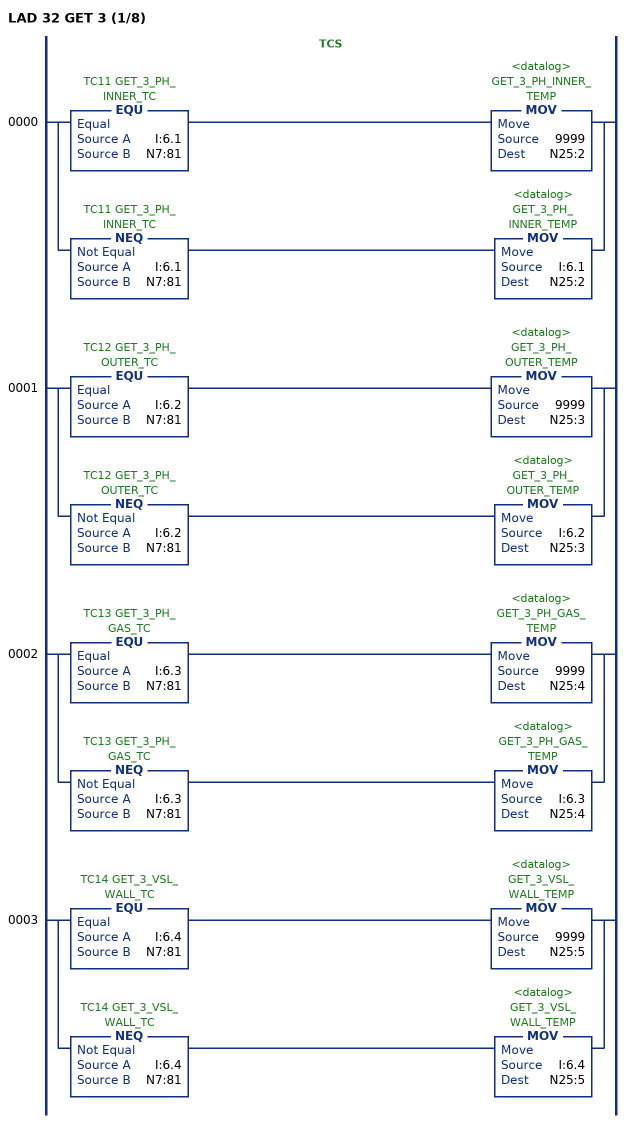
% Rung: 0 %
% TITLE: TCS %
SOR BST EQU I:6.1 N7:81 MOV 9999 N25:2 NXB NEQ I:6.1 N7:81 MOV I:6.1 N25:2 BND EOR
%   I:6.1  GET_3_PH_INNER_TC  "TC11" %
%   N7:81  TC_OPEN_SP  "CONFIG The value read by an open TC input" %
%   N25:2  GET_3_PH_INNER_TEMP  "<datalog>" %
% Rung: 1 %
SOR BST EQU I:6.2 N7:81 MOV 9999 N25:3 NXB NEQ I:6.2 N7:81 MOV I:6.2 N25:3 BND EOR
%   I:6.2  GET_3_PH_OUTER_TC  "TC12" %
%   N7:81  TC_OPEN_SP  "CONFIG The value read by an open TC input" %
%   N25:3  GET_3_PH_OUTER_TEMP  "<datalog>" %
% Rung: 2 %
SOR BST EQU I:6.3 N7:81 MOV 9999 N25:4 NXB NEQ I:6.3 N7:81 MOV I:6.3 N25:4 BND EOR
%   I:6.3  GET_3_PH_GAS_TC  "TC13" %
%   N7:81  TC_OPEN_SP  "CONFIG The value read by an open TC input" %
%   N25:4  GET_3_PH_GAS_TEMP  "<datalog>" %
% Rung: 3 %
SOR BST EQU I:6.4 N7:81 MOV 9999 N25:5 NXB NEQ I:6.4 N7:81 MOV I:6.4 N25:5 BND EOR
%   I:6.4  GET_3_VSL_WALL_TC  "TC14" %
%   N7:81  TC_OPEN_SP  "CONFIG The value read by an open TC input" %
%   N25:5  GET_3_VSL_WALL_TEMP  "<datalog>" %

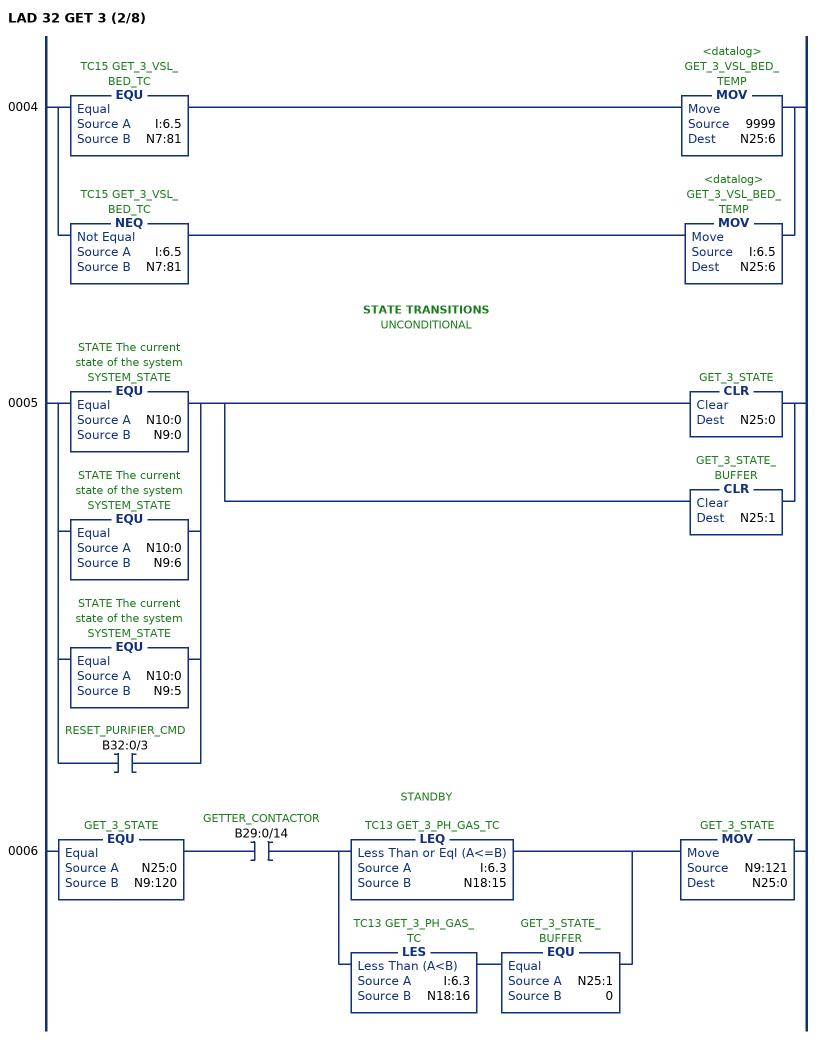
% Rung: 4 %
SOR BST EQU I:6.5 N7:81 MOV 9999 N25:6 NXB NEQ I:6.5 N7:81 MOV I:6.5 N25:6 BND EOR
%   I:6.5  GET_3_VSL_BED_TC  "TC15" %
%   N7:81  TC_OPEN_SP  "CONFIG The value read by an open TC input" %
%   N25:6  GET_3_VSL_BED_TEMP  "<datalog>" %
% Rung: 5 %
% TITLE: STATE TRANSITIONS %
% UNCONDITIONAL %
SOR BST EQU N10:0 N9:0 NXB EQU N10:0 N9:6 NXB EQU N10:0 N9:5 NXB XIC B32:0/3 BND BST CLR N25:0 NXB CLR N25:1 BND EOR
%   N10:0  SYSTEM_STATE  "STATE The current state of the system" %
%   N9:0  SYSTEM_OFFLINE %
%   N9:6  SYSTEM_PURGE %
%   N9:5  SYSTEM_QUICK_START %
%   B32:0/3  RESET_PURIFIER_CMD %
%   N25:0  GET_3_STATE %
%   N25:1  GET_3_STATE_BUFFER %
% Rung: 6 %
% STANDBY %
SOR EQU N25:0 N9:120 XIC B29:0/14 BST LEQ I:6.3 N18:15 NXB LES I:6.3 N18:16 EQU N25:1 0 BND MOV N9:121 N25:0 EOR
%   N25:0  GET_3_STATE %
%   N9:120  GETTER_STANDBY %
%   B29:0/14  GETTER_CONTACTOR %
%   I:6.3  GET_3_PH_GAS_TC  "TC13" %
%   N18:15  GETTER_SS_BEGIN_TEMP %
%   N18:16  GETTER_SS_END_TEMP %
%   N25:1  GET_3_STATE_BUFFER %
%   N9:121  GETTER_SOFTSTART %

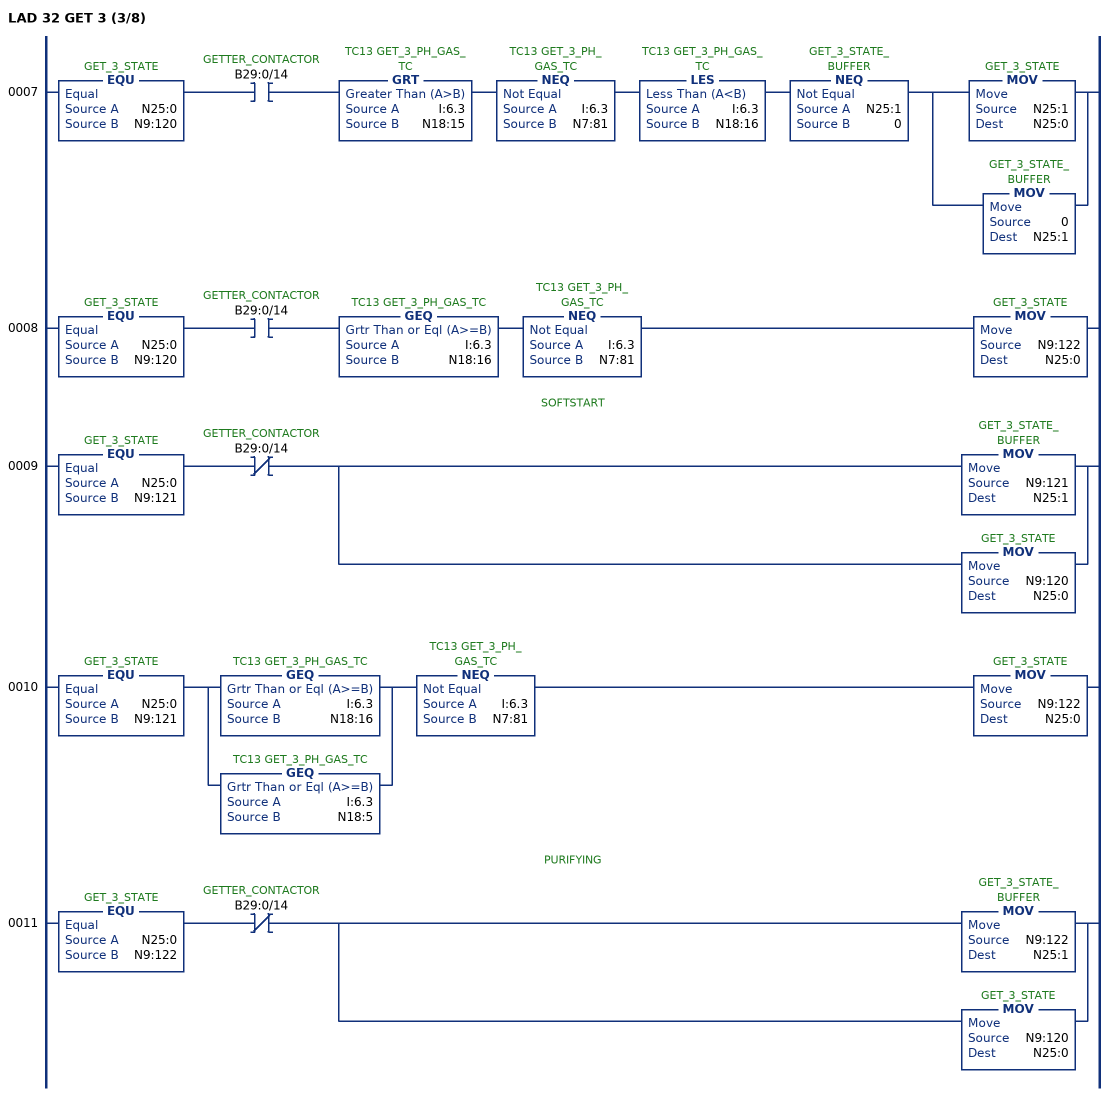
% Rung: 7 %
SOR EQU N25:0 N9:120 XIC B29:0/14 GRT I:6.3 N18:15 NEQ I:6.3 N7:81 LES I:6.3 N18:16 NEQ N25:1 0 BST MOV N25:1 N25:0 NXB MOV 0 N25:1 BND EOR
%   N25:0  GET_3_STATE %
%   N9:120  GETTER_STANDBY %
%   B29:0/14  GETTER_CONTACTOR %
%   I:6.3  GET_3_PH_GAS_TC  "TC13" %
%   N18:15  GETTER_SS_BEGIN_TEMP %
%   N7:81  TC_OPEN_SP  "CONFIG The value read by an open TC input" %
%   N18:16  GETTER_SS_END_TEMP %
%   N25:1  GET_3_STATE_BUFFER %
% Rung: 8 %
SOR EQU N25:0 N9:120 XIC B29:0/14 GEQ I:6.3 N18:16 NEQ I:6.3 N7:81 MOV N9:122 N25:0 EOR
%   N25:0  GET_3_STATE %
%   N9:120  GETTER_STANDBY %
%   B29:0/14  GETTER_CONTACTOR %
%   I:6.3  GET_3_PH_GAS_TC  "TC13" %
%   N18:16  GETTER_SS_END_TEMP %
%   N7:81  TC_OPEN_SP  "CONFIG The value read by an open TC input" %
%   N9:122  GETTER_PURIFYING %
% Rung: 9 %
% SOFTSTART %
SOR EQU N25:0 N9:121 XIO B29:0/14 BST MOV N9:121 N25:1 NXB MOV N9:120 N25:0 BND EOR
%   N25:0  GET_3_STATE %
%   N9:121  GETTER_SOFTSTART %
%   B29:0/14  GETTER_CONTACTOR %
%   N25:1  GET_3_STATE_BUFFER %
%   N9:120  GETTER_STANDBY %
% Rung: 10 %
SOR EQU N25:0 N9:121 BST GEQ I:6.3 N18:16 NXB GEQ I:6.3 N18:5 BND NEQ I:6.3 N7:81 MOV N9:122 N25:0 EOR
%   N25:0  GET_3_STATE %
%   N9:121  GETTER_SOFTSTART %
%   I:6.3  GET_3_PH_GAS_TC  "TC13" %
%   N18:16  GETTER_SS_END_TEMP %
%   N18:5  GETTER_PH_SP  "<datalog>" %
%   N7:81  TC_OPEN_SP  "CONFIG The value read by an open TC input" %
%   N9:122  GETTER_PURIFYING %
% Rung: 11 %
% PURIFYING %
SOR EQU N25:0 N9:122 XIO B29:0/14 BST MOV N9:122 N25:1 NXB MOV N9:120 N25:0 BND EOR
%   N25:0  GET_3_STATE %
%   N9:122  GETTER_PURIFYING %
%   B29:0/14  GETTER_CONTACTOR %
%   N25:1  GET_3_STATE_BUFFER %
%   N9:120  GETTER_STANDBY %

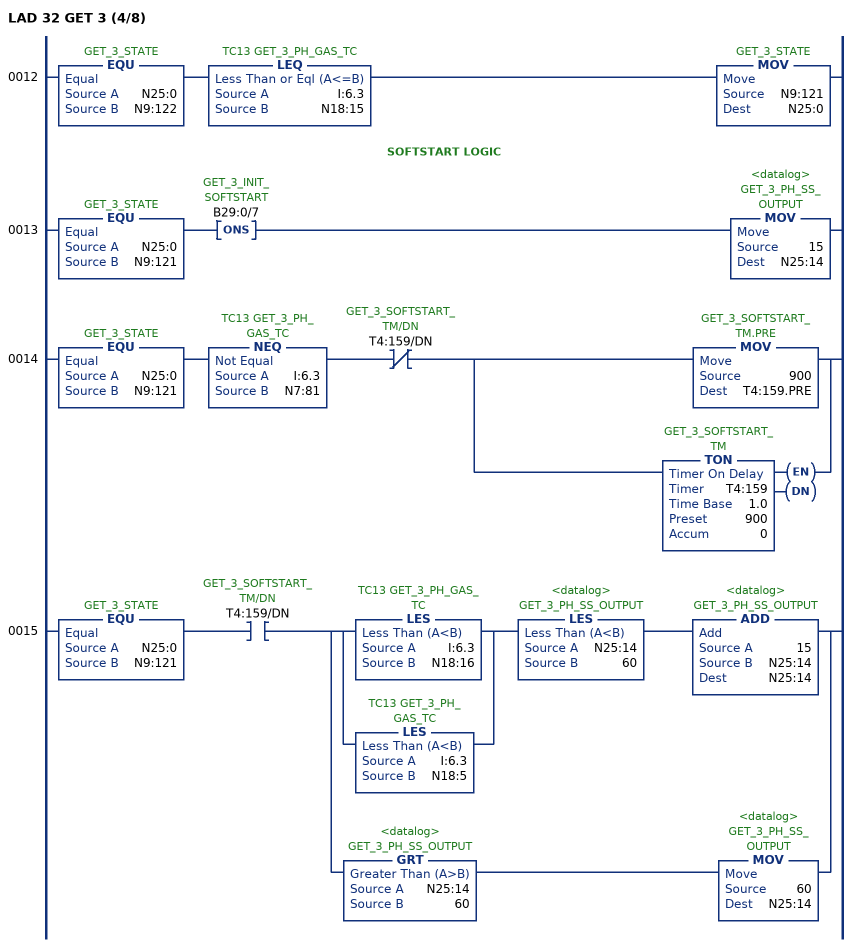
% Rung: 12 %
SOR EQU N25:0 N9:122 LEQ I:6.3 N18:15 MOV N9:121 N25:0 EOR
%   N25:0  GET_3_STATE %
%   N9:122  GETTER_PURIFYING %
%   I:6.3  GET_3_PH_GAS_TC  "TC13" %
%   N18:15  GETTER_SS_BEGIN_TEMP %
%   N9:121  GETTER_SOFTSTART %
% Rung: 13 %
% TITLE: SOFTSTART LOGIC %
SOR EQU N25:0 N9:121 ONS B29:0/7 MOV 15 N25:14 EOR
%   N25:0  GET_3_STATE %
%   N9:121  GETTER_SOFTSTART %
%   B29:0/7  GET_3_INIT_SOFTSTART %
%   N25:14  GET_3_PH_SS_OUTPUT  "<datalog>" %
% Rung: 14 %
SOR EQU N25:0 N9:121 NEQ I:6.3 N7:81 XIO T4:159/DN BST MOV 900 T4:159.PRE NXB TON T4:159 1.0 900 0 BND EOR
%   N25:0  GET_3_STATE %
%   N9:121  GETTER_SOFTSTART %
%   I:6.3  GET_3_PH_GAS_TC  "TC13" %
%   N7:81  TC_OPEN_SP  "CONFIG The value read by an open TC input" %
%   T4:159  GET_3_SOFTSTART_TM %
% Rung: 15 %
SOR EQU N25:0 N9:121 XIC T4:159/DN BST BST LES I:6.3 N18:16 NXB LES I:6.3 N18:5 BND LES N25:14 60 ADD 15 N25:14 N25:14 NXB GRT N25:14 60 MOV 60 N25:14 BND EOR
%   N25:0  GET_3_STATE %
%   N9:121  GETTER_SOFTSTART %
%   T4:159  GET_3_SOFTSTART_TM %
%   I:6.3  GET_3_PH_GAS_TC  "TC13" %
%   N18:16  GETTER_SS_END_TEMP %
%   N18:5  GETTER_PH_SP  "<datalog>" %
%   N25:14  GET_3_PH_SS_OUTPUT  "<datalog>" %

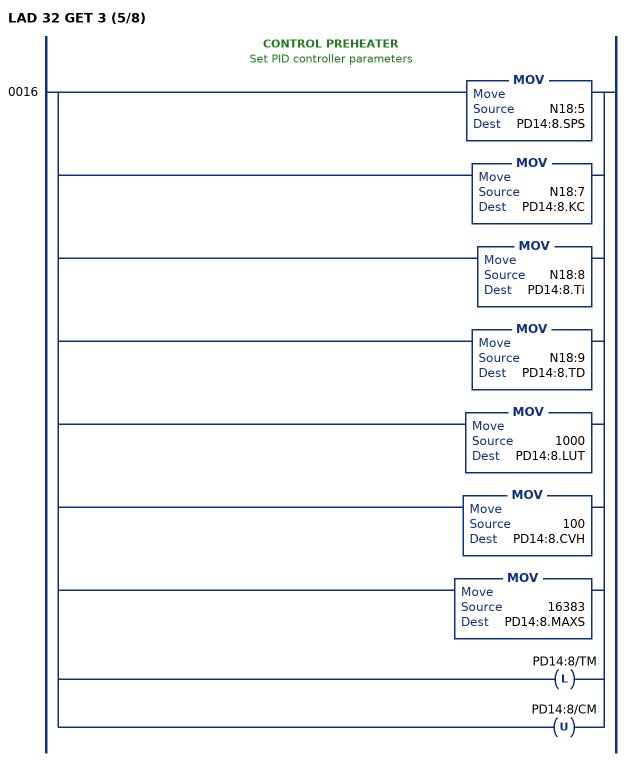
% Rung: 16 %
% TITLE: CONTROL PREHEATER %
% Set PID controller parameters %
SOR BST MOV N18:5 PD14:8.SPS NXB MOV N18:7 PD14:8.KC NXB MOV N18:8 PD14:8.Ti NXB MOV N18:9 PD14:8.TD NXB MOV 1000 PD14:8.LUT NXB MOV 100 PD14:8.CVH NXB MOV 16383 PD14:8.MAXS NXB OTL PD14:8/TM NXB OTU PD14:8/CM BND EOR
%   N18:5  GETTER_PH_SP  "<datalog>" %
%   N18:7  GET_PH_PID_GAIN %
%   N18:8  GET_PH_PID_INTEG %
%   N18:9  GET_PH_PID_DERIV %

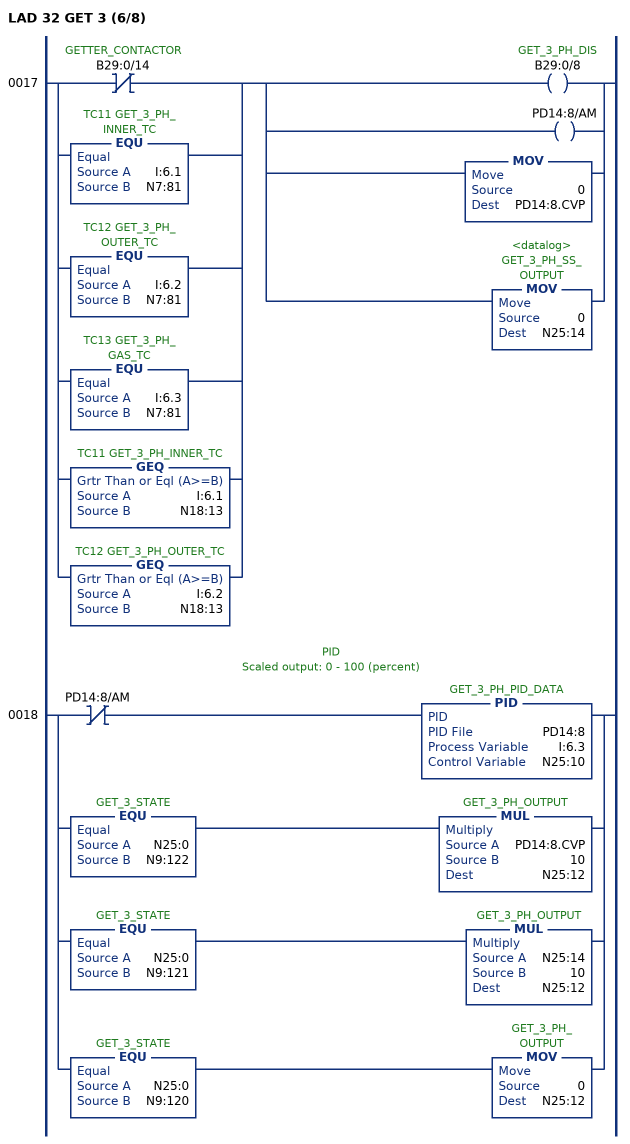
% Rung: 17 %
SOR BST XIO B29:0/14 NXB EQU I:6.1 N7:81 NXB EQU I:6.2 N7:81 NXB EQU I:6.3 N7:81 NXB GEQ I:6.1 N18:13 NXB GEQ I:6.2 N18:13 BND BST OTE B29:0/8 NXB OTE PD14:8/AM NXB MOV 0 PD14:8.CVP NXB MOV 0 N25:14 BND EOR
%   B29:0/14  GETTER_CONTACTOR %
%   I:6.1  GET_3_PH_INNER_TC  "TC11" %
%   N7:81  TC_OPEN_SP  "CONFIG The value read by an open TC input" %
%   I:6.2  GET_3_PH_OUTER_TC  "TC12" %
%   I:6.3  GET_3_PH_GAS_TC  "TC13" %
%   N18:13  GET_PH_ROD_LIMIT %
%   B29:0/8  GET_3_PH_DIS %
%   N25:14  GET_3_PH_SS_OUTPUT  "<datalog>" %
% Rung: 18 %
% PID
% Scaled output: 0 - 100 (percent) %
SOR BST XIO PD14:8/AM PID PD14:8 I:6.3 N25:10 NXB EQU N25:0 N9:122 MUL PD14:8.CVP 10 N25:12 NXB EQU N25:0 N9:121 MUL N25:14 10 N25:12 NXB EQU N25:0 N9:120 MOV 0 N25:12 BND EOR
%   PD14:8  GET_3_PH_PID_DATA %
%   I:6.3  GET_3_PH_GAS_TC  "TC13" %
%   N25:10  GET_3_PH_OUT_RAW %
%   N25:0  GET_3_STATE %
%   N9:122  GETTER_PURIFYING %
%   N25:12  GET_3_PH_OUTPUT %
%   N9:121  GETTER_SOFTSTART %
%   N25:14  GET_3_PH_SS_OUTPUT  "<datalog>" %
%   N9:120  GETTER_STANDBY %

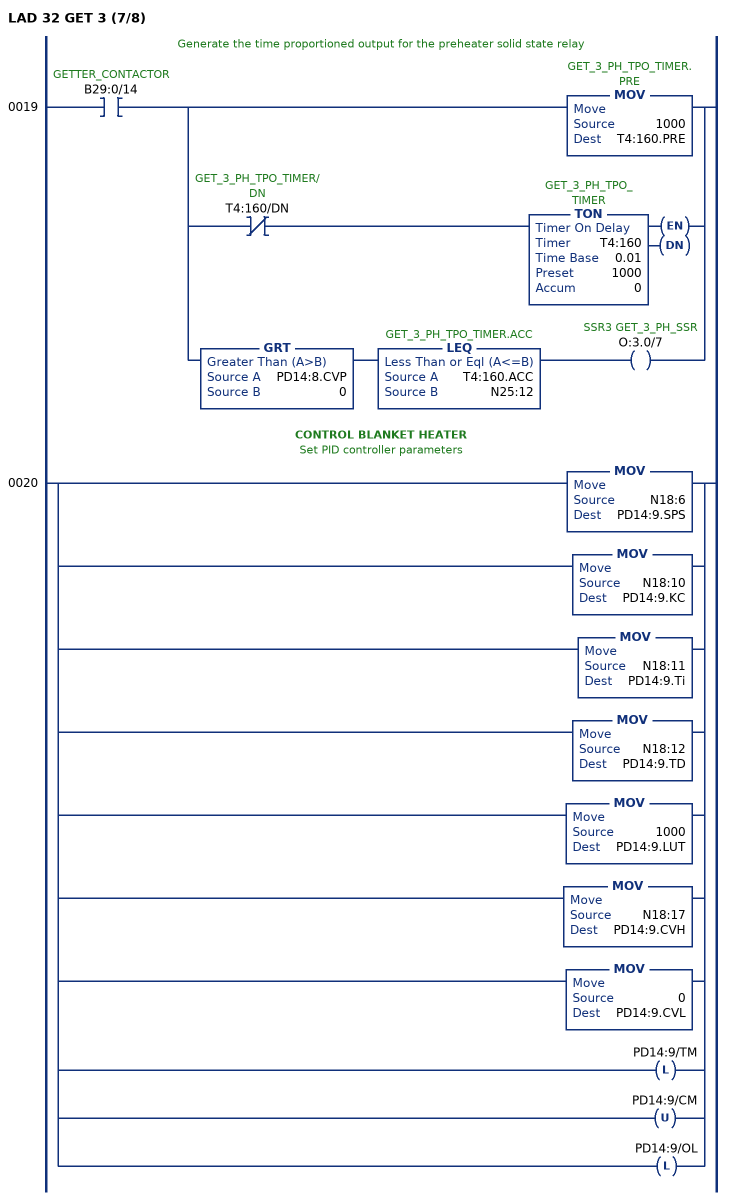
% Rung: 19 %
% Generate the time proportioned output for the preheater solid state relay %
SOR XIC B29:0/14 BST MOV 1000 T4:160.PRE NXB XIO T4:160/DN TON T4:160 0.01 1000 0 NXB GRT PD14:8.CVP 0 LEQ T4:160.ACC N25:12 OTE O:3.0/7 BND EOR
%   B29:0/14  GETTER_CONTACTOR %
%   T4:160  GET_3_PH_TPO_TIMER %
%   N25:12  GET_3_PH_OUTPUT %
%   O:3.0/7  GET_3_PH_SSR  "SSR3" %
% Rung: 20 %
% TITLE: CONTROL BLANKET HEATER %
% Set PID controller parameters %
SOR BST MOV N18:6 PD14:9.SPS NXB MOV N18:10 PD14:9.KC NXB MOV N18:11 PD14:9.Ti NXB MOV N18:12 PD14:9.TD NXB MOV 1000 PD14:9.LUT NXB MOV N18:17 PD14:9.CVH NXB MOV 0 PD14:9.CVL NXB OTL PD14:9/TM NXB OTU PD14:9/CM NXB OTL PD14:9/OL BND EOR
%   N18:6  GETTER_BLKT_SP  "<datalog>" %
%   N18:10  GET_BLKT_PID_GAIN %
%   N18:11  GET_BLKT_PID_INTEG %
%   N18:12  GET_BLKT_PID_DERIV %
%   N18:17  GET_BLKT_PID_HI_LIM %

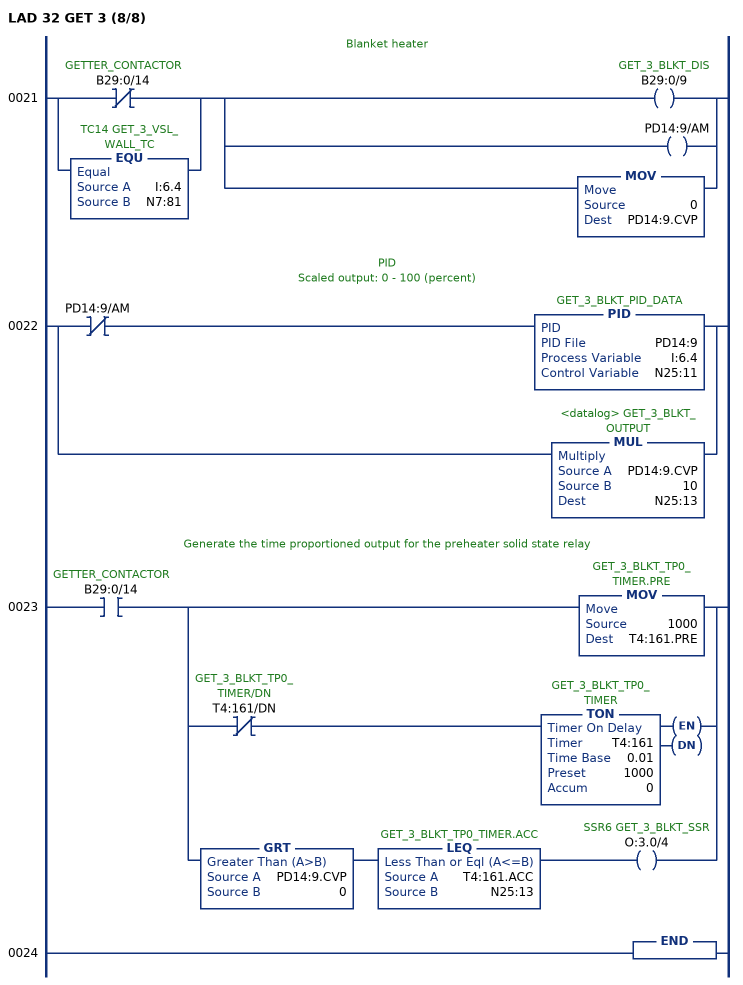
% Rung: 21 %
% Blanket heater %
SOR BST XIO B29:0/14 NXB EQU I:6.4 N7:81 BND BST OTE B29:0/9 NXB OTE PD14:9/AM NXB MOV 0 PD14:9.CVP BND EOR
%   B29:0/14  GETTER_CONTACTOR %
%   I:6.4  GET_3_VSL_WALL_TC  "TC14" %
%   N7:81  TC_OPEN_SP  "CONFIG The value read by an open TC input" %
%   B29:0/9  GET_3_BLKT_DIS %
% Rung: 22 %
% PID
% Scaled output: 0 - 100 (percent) %
SOR BST XIO PD14:9/AM PID PD14:9 I:6.4 N25:11 NXB MUL PD14:9.CVP 10 N25:13 BND EOR
%   PD14:9  GET_3_BLKT_PID_DATA %
%   I:6.4  GET_3_VSL_WALL_TC  "TC14" %
%   N25:11  GET_3_BLKT_OUT_RAW %
%   N25:13  GET_3_BLKT_OUTPUT  "<datalog>" %
% Rung: 23 %
% Generate the time proportioned output for the preheater solid state relay %
SOR XIC B29:0/14 BST MOV 1000 T4:161.PRE NXB XIO T4:161/DN TON T4:161 0.01 1000 0 NXB GRT PD14:9.CVP 0 LEQ T4:161.ACC N25:13 OTE O:3.0/4 BND EOR
%   B29:0/14  GETTER_CONTACTOR %
%   T4:161  GET_3_BLKT_TP0_TIMER %
%   N25:13  GET_3_BLKT_OUTPUT  "<datalog>" %
%   O:3.0/4  GET_3_BLKT_SSR  "SSR6" %
% Rung: 24 %
SOR END EOR

LADDER 49 "MODBUS"
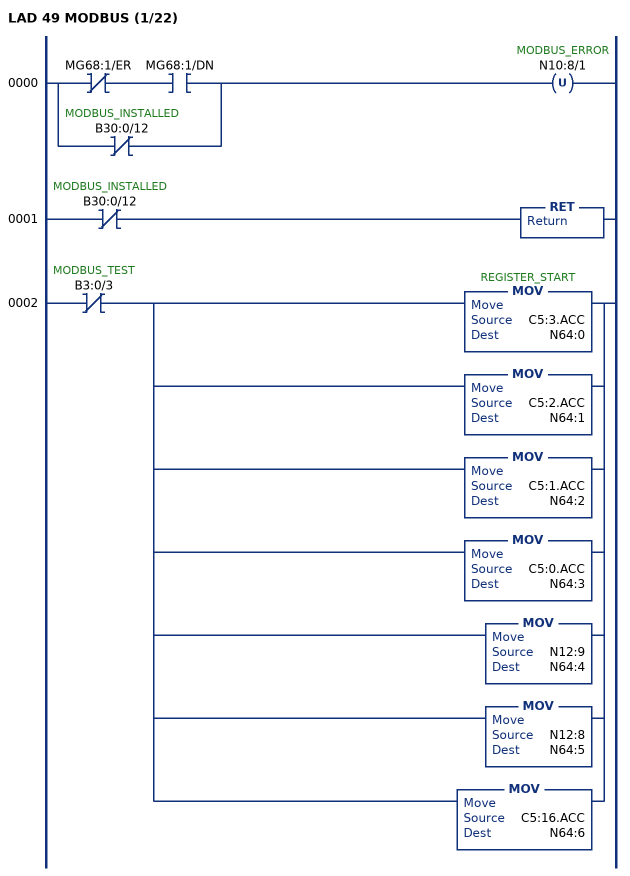
% Rung: 0 %
SOR BST XIO MG68:1/ER XIC MG68:1/DN NXB XIO B30:0/12 BND OTU N10:8/1 EOR
%   B30:0/12  MODBUS_INSTALLED %
%   N10:8/1  MODBUS_ERROR %
% Rung: 1 %
SOR XIO B30:0/12 RET EOR
%   B30:0/12  MODBUS_INSTALLED %
% Rung: 2 %
SOR XIO B3:0/3 BST MOV C5:3.ACC N64:0 NXB MOV C5:2.ACC N64:1 NXB MOV C5:1.ACC N64:2 NXB MOV C5:0.ACC N64:3 NXB MOV N12:9 N64:4 NXB MOV N12:8 N64:5 NXB MOV C5:16.ACC N64:6 BND EOR
%   B3:0/3  MODBUS_TEST %
%   C5:3  PURIFY_ACTIVE_TTL_DY  "COUNTER The number of total elapsed purification days for the process equipment" %
%   N64:0  REGISTER_START %
%   C5:2  PURIFY_ACTIVE_TTL_HR  "COUNTER The number of total elapsed purification hours for the process equipment" %
%   C5:1  PURIFY_ACTIVE_MINUTE  "COUNTER The number of elapsed purification minutes for the current ADS (60 min)" %
%   C5:0  PURIFY_ACTIVE_HOURS  "COUNTER The number of elapsed purification hours for the current ADS" %
%   N12:9  MIN_LEFT_IN_PURIFY %
%   N12:8  HRS_LEFT_IN_PURIFY %
%   C5:16  GETTER_SERVICE_DAYS %

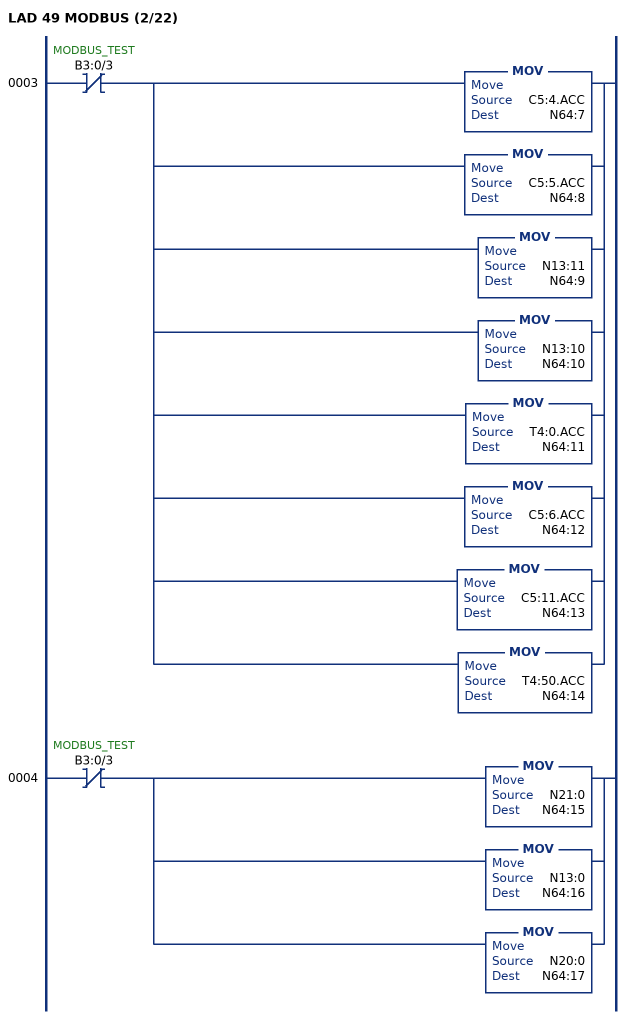
% Rung: 3 %
SOR XIO B3:0/3 BST MOV C5:4.ACC N64:7 NXB MOV C5:5.ACC N64:8 NXB MOV N13:11 N64:9 NXB MOV N13:10 N64:10 NXB MOV T4:0.ACC N64:11 NXB MOV C5:6.ACC N64:12 NXB MOV C5:11.ACC N64:13 NXB MOV T4:50.ACC N64:14 BND EOR
%   B3:0/3  MODBUS_TEST %
%   C5:4  REGEN_RUN_MINUTE %
%   C5:5  REGEN_COOL_MINUTE  "COUNTER Regen the number of minutes for which the bed has cooled" %
%   N13:11  REGEN_MIN_LEFT  "STATUS Preheater Alarm Measured temperature change" %
%   N13:10  REGEN_HRS_LEFT  "STATUS Regen Preheater Temperature Initial Temperature" %
%   T4:0  PURIFY_OVERLAP_TIMER  "TIMER Purify Overlap" %
%   C5:6  START_PURGE_CTR %
%   C5:11  H2_LEAK_RST_MIN %
%   T4:50  H2_LEAK_RST_SEC %
% Rung: 4 %
SOR XIO B3:0/3 BST MOV N21:0 N64:15 NXB MOV N13:0 N64:16 NXB MOV N20:0 N64:17 BND EOR
%   B3:0/3  MODBUS_TEST %
%   N21:0  START_STATE %
%   N13:0  REGEN_STATE  "STATE The current state of the regen process" %
%   N20:0  PURGE_STATE %

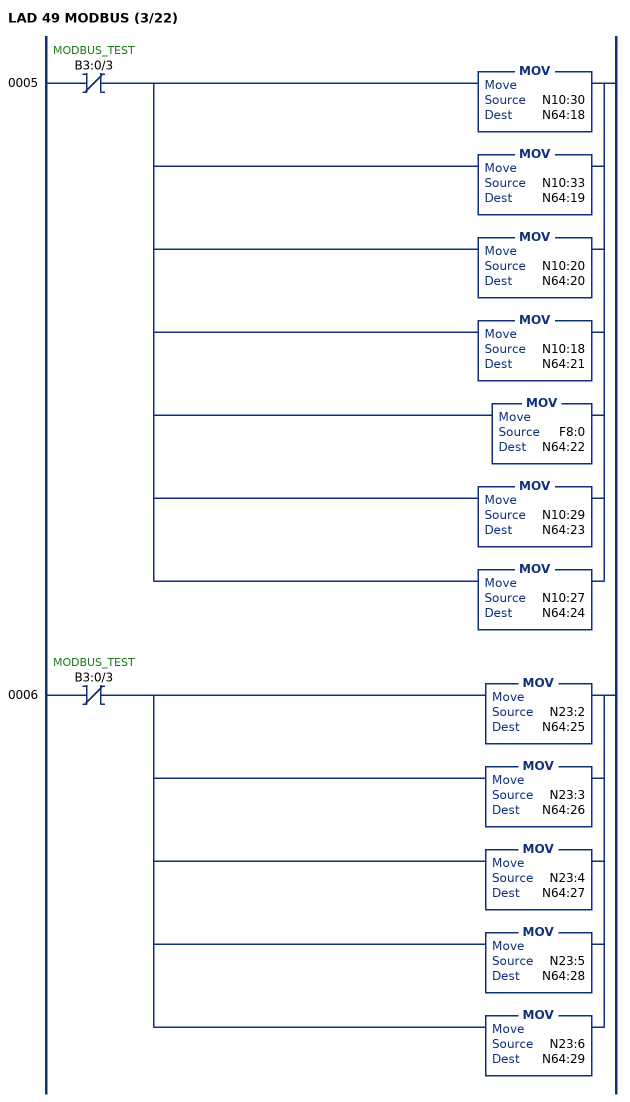
% Rung: 5 %
SOR XIO B3:0/3 BST MOV N10:30 N64:18 NXB MOV N10:33 N64:19 NXB MOV N10:20 N64:20 NXB MOV N10:18 N64:21 NXB MOV F8:0 N64:22 NXB MOV N10:29 N64:23 NXB MOV N10:27 N64:24 BND EOR
%   B3:0/3  MODBUS_TEST %
%   N10:30  ADS_A_INLET_PX_PSIG %
%   N10:33  ADS_B_INLET_PX_PSIG %
%   N10:20  OUTLET_PX_PSIG %
%   N10:18  INLET_PX_PSIG %
%   F8:0  MFM_CUM_HR %
%   N10:29  MFC_SLPM %
%   N10:27  MFC_SETPOINT %
% Rung: 6 %
SOR XIO B3:0/3 BST MOV N23:2 N64:25 NXB MOV N23:3 N64:26 NXB MOV N23:4 N64:27 NXB MOV N23:5 N64:28 NXB MOV N23:6 N64:29 BND EOR
%   B3:0/3  MODBUS_TEST %
%   N23:2  GET_1_PH_INNER_TEMP  "<datalog>" %
%   N23:3  GET_1_PH_OUTER_TEMP  "<datalog>" %
%   N23:4  GET_1_PH_GAS_TEMP  "<datalog>" %
%   N23:5  GET_1_VSL_WALL_TEMP  "<datalog>" %
%   N23:6  GET_1_VSL_BED_TEMP  "<datalog>" %

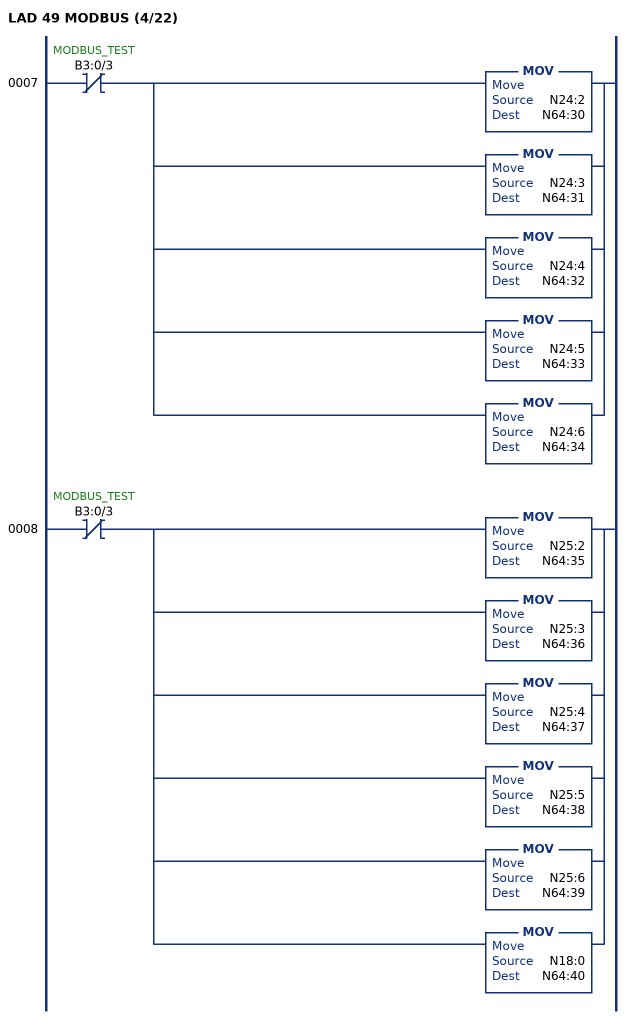
% Rung: 7 %
SOR XIO B3:0/3 BST MOV N24:2 N64:30 NXB MOV N24:3 N64:31 NXB MOV N24:4 N64:32 NXB MOV N24:5 N64:33 NXB MOV N24:6 N64:34 BND EOR
%   B3:0/3  MODBUS_TEST %
%   N24:2  GET_2_PH_INNER_TEMP  "<datalog>" %
%   N24:3  GET_2_PH_OUTER_TEMP  "<datalog>" %
%   N24:4  GET_2_PH_GAS_TEMP  "<datalog>" %
%   N24:5  GET_2_VSL_WALL_TEMP  "<datalog>" %
%   N24:6  GET_2_VSL_BED_TEMP  "<datalog>" %
% Rung: 8 %
SOR XIO B3:0/3 BST MOV N25:2 N64:35 NXB MOV N25:3 N64:36 NXB MOV N25:4 N64:37 NXB MOV N25:5 N64:38 NXB MOV N25:6 N64:39 NXB MOV N18:0 N64:40 BND EOR
%   B3:0/3  MODBUS_TEST %
%   N25:2  GET_3_PH_INNER_TEMP  "<datalog>" %
%   N25:3  GET_3_PH_OUTER_TEMP  "<datalog>" %
%   N25:4  GET_3_PH_GAS_TEMP  "<datalog>" %
%   N25:5  GET_3_VSL_WALL_TEMP  "<datalog>" %
%   N25:6  GET_3_VSL_BED_TEMP  "<datalog>" %
%   N18:0  GET_VSL_OUT_GAS_TEMP %

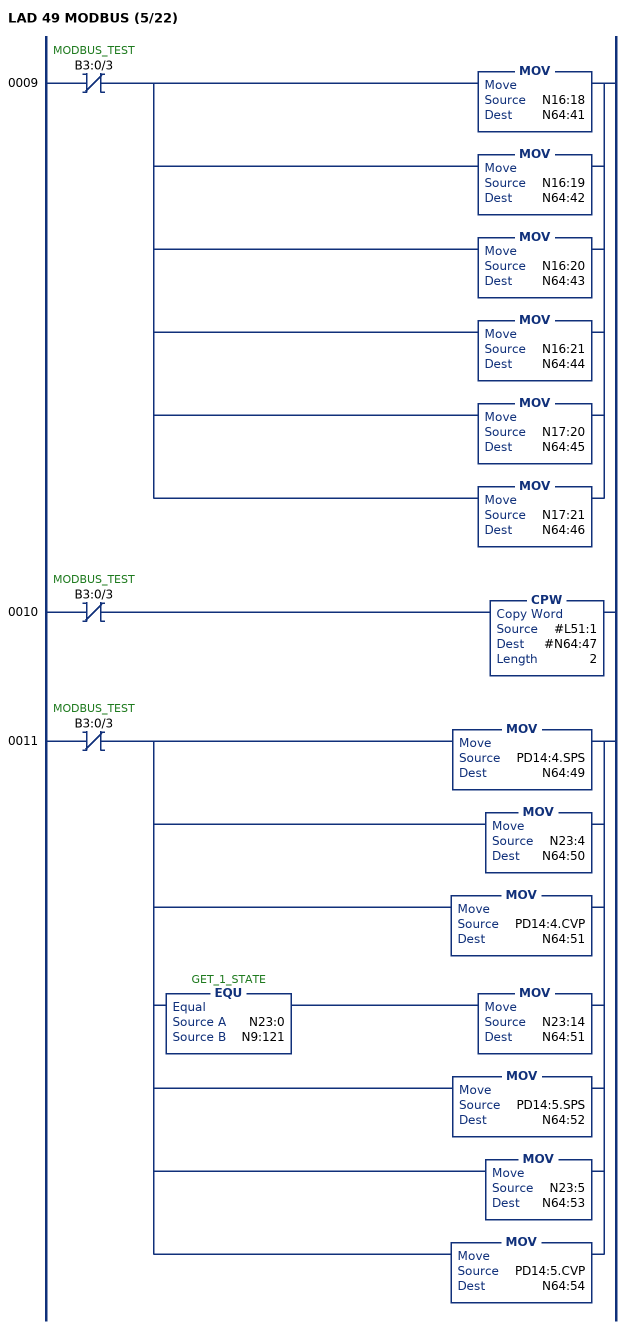
% Rung: 9 %
SOR XIO B3:0/3 BST MOV N16:18 N64:41 NXB MOV N16:19 N64:42 NXB MOV N16:20 N64:43 NXB MOV N16:21 N64:44 NXB MOV N17:20 N64:45 NXB MOV N17:21 N64:46 BND EOR
%   B3:0/3  MODBUS_TEST %
%   N16:18  ADS_PH_GAS_TEMP_READ  "<datalog>" %
%   N16:19  ADS_PH_ROD_TEMP_READ  "<datalog>" %
%   N16:20  ADS_A_WALL_TEMP_READ  "<datalog>" %
%   N16:21  ADS_A_BED_TEMP_READ  "<datalog>" %
%   N17:20  ADS_B_WALL_TEMP_READ  "<datalog>" %
%   N17:21  ADS_B_BED_TEMP_READ  "<datalog>" %
% Rung: 10 %
SOR XIO B3:0/3 CPW #L51:1 #N64:47 2 EOR
%   B3:0/3  MODBUS_TEST %
%   L51:1  TOTAL_FLOW_MODBUS %
% Rung: 11 %
SOR XIO B3:0/3 BST MOV PD14:4.SPS N64:49 NXB MOV N23:4 N64:50 NXB BST MOV PD14:4.CVP N64:51 NXB EQU N23:0 N9:121 MOV N23:14 N64:51 BND NXB MOV PD14:5.SPS N64:52 NXB MOV N23:5 N64:53 NXB MOV PD14:5.CVP N64:54 BND EOR
%   B3:0/3  MODBUS_TEST %
%   N23:4  GET_1_PH_GAS_TEMP  "<datalog>" %
%   N23:0  GET_1_STATE %
%   N9:121  GETTER_SOFTSTART %
%   N23:14  GET_1_PH_SS_OUTPUT %
%   N23:5  GET_1_VSL_WALL_TEMP  "<datalog>" %

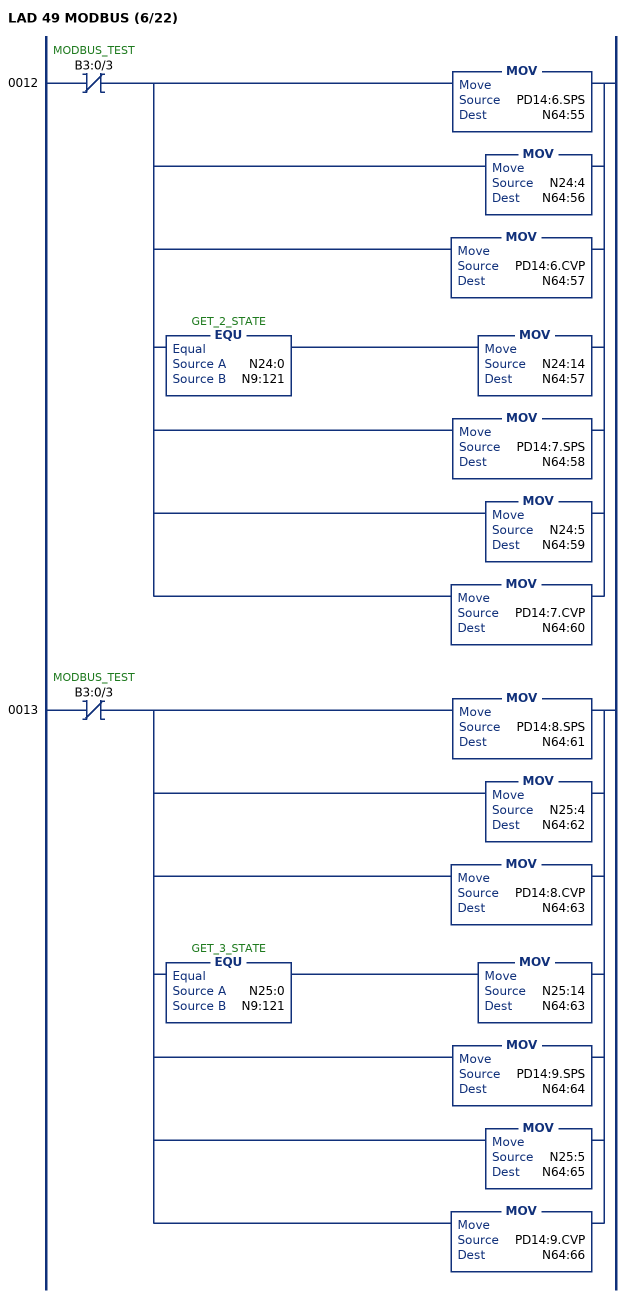
% Rung: 12 %
SOR XIO B3:0/3 BST MOV PD14:6.SPS N64:55 NXB MOV N24:4 N64:56 NXB BST MOV PD14:6.CVP N64:57 NXB EQU N24:0 N9:121 MOV N24:14 N64:57 BND NXB MOV PD14:7.SPS N64:58 NXB MOV N24:5 N64:59 NXB MOV PD14:7.CVP N64:60 BND EOR
%   B3:0/3  MODBUS_TEST %
%   N24:4  GET_2_PH_GAS_TEMP  "<datalog>" %
%   N24:0  GET_2_STATE %
%   N9:121  GETTER_SOFTSTART %
%   N24:14  GET_2_PH_SS_OUTPUT %
%   N24:5  GET_2_VSL_WALL_TEMP  "<datalog>" %
% Rung: 13 %
SOR XIO B3:0/3 BST MOV PD14:8.SPS N64:61 NXB MOV N25:4 N64:62 NXB BST MOV PD14:8.CVP N64:63 NXB EQU N25:0 N9:121 MOV N25:14 N64:63 BND NXB MOV PD14:9.SPS N64:64 NXB MOV N25:5 N64:65 NXB MOV PD14:9.CVP N64:66 BND EOR
%   B3:0/3  MODBUS_TEST %
%   N25:4  GET_3_PH_GAS_TEMP  "<datalog>" %
%   N25:0  GET_3_STATE %
%   N9:121  GETTER_SOFTSTART %
%   N25:14  GET_3_PH_SS_OUTPUT  "<datalog>" %
%   N25:5  GET_3_VSL_WALL_TEMP  "<datalog>" %

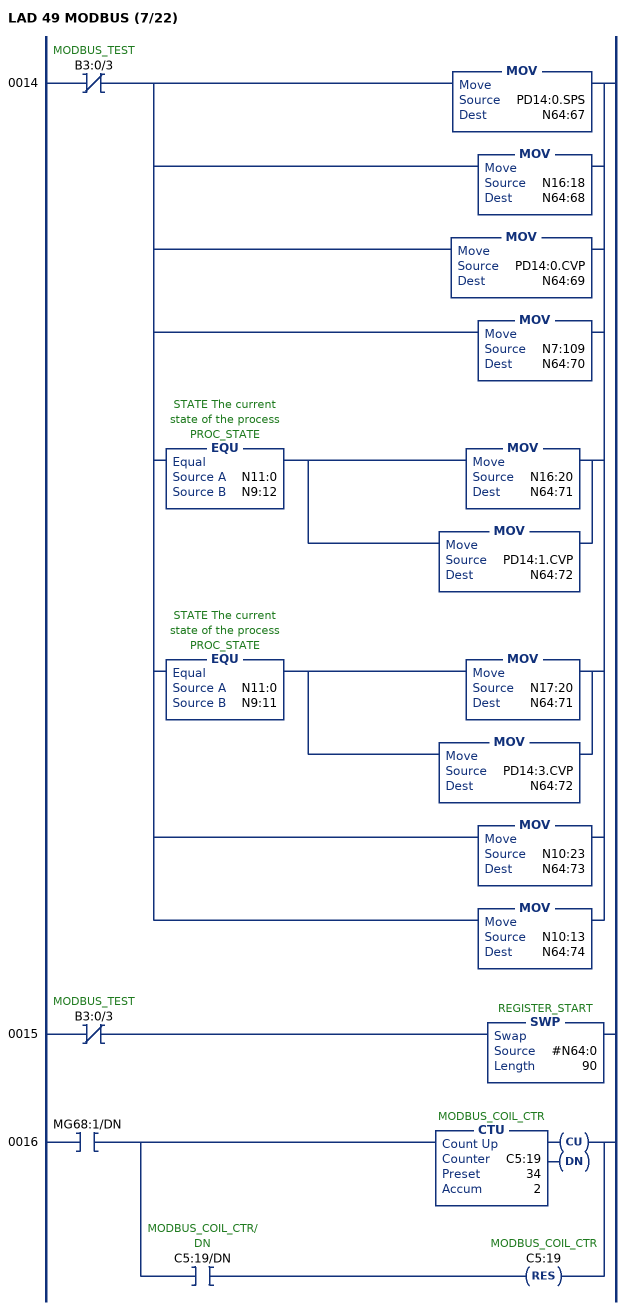
% Rung: 14 %
SOR XIO B3:0/3 BST MOV PD14:0.SPS N64:67 NXB MOV N16:18 N64:68 NXB MOV PD14:0.CVP N64:69 NXB MOV N7:109 N64:70 NXB EQU N11:0 N9:12 BST MOV N16:20 N64:71 NXB MOV PD14:1.CVP N64:72 BND NXB EQU N11:0 N9:11 BST MOV N17:20 N64:71 NXB MOV PD14:3.CVP N64:72 BND NXB MOV N10:23 N64:73 NXB MOV N10:13 N64:74 BND EOR
%   B3:0/3  MODBUS_TEST %
%   N16:18  ADS_PH_GAS_TEMP_READ  "<datalog>" %
%   N7:109  BLANKET_SP  "<datalog> CONTROL Blanket PID Setpoint" %
%   N11:0  PROC_STATE  "STATE The current state of the process" %
%   N9:12  PROC_PFY_B_REG_A  "STATE Process Purify B" %
%   N16:20  ADS_A_WALL_TEMP_READ  "<datalog>" %
%   N9:11  PROC_PFY_A_REG_B  "STATE Process Purify A" %
%   N17:20  ADS_B_WALL_TEMP_READ  "<datalog>" %
%   N10:23  H2_LEVEL_PERCENT %
%   N10:13  DIFF_PRES_TRANS_READ %
% Rung: 15 %
SOR XIO B3:0/3 SWP #N64:0 90 EOR
%   B3:0/3  MODBUS_TEST %
%   N64:0  REGISTER_START %
% Rung: 16 %
SOR XIC MG68:1/DN BST CTU C5:19 34 2 NXB XIC C5:19/DN RES C5:19 BND EOR
%   C5:19  MODBUS_COIL_CTR %

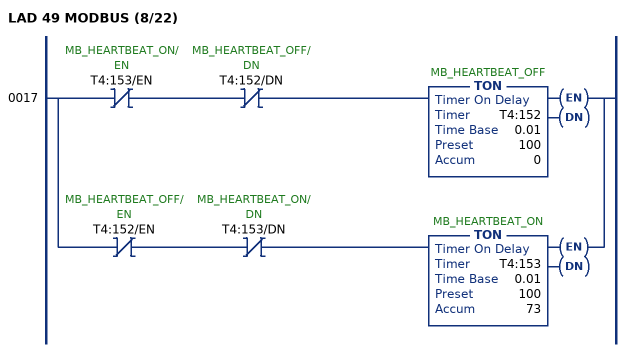
% Rung: 17 %
SOR BST XIO T4:153/EN XIO T4:152/DN TON T4:152 0.01 100 0 NXB XIO T4:152/EN XIO T4:153/DN TON T4:153 0.01 100 73 BND EOR
%   T4:153  MB_HEARTBEAT_ON %
%   T4:152  MB_HEARTBEAT_OFF %

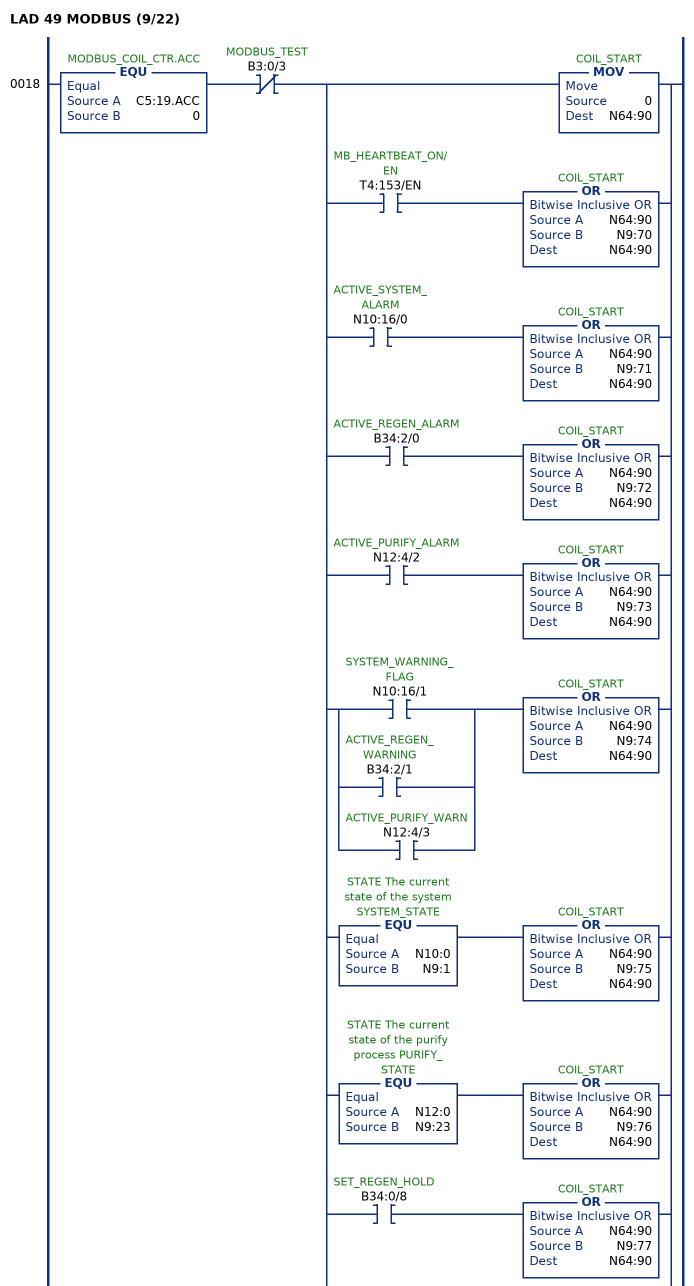

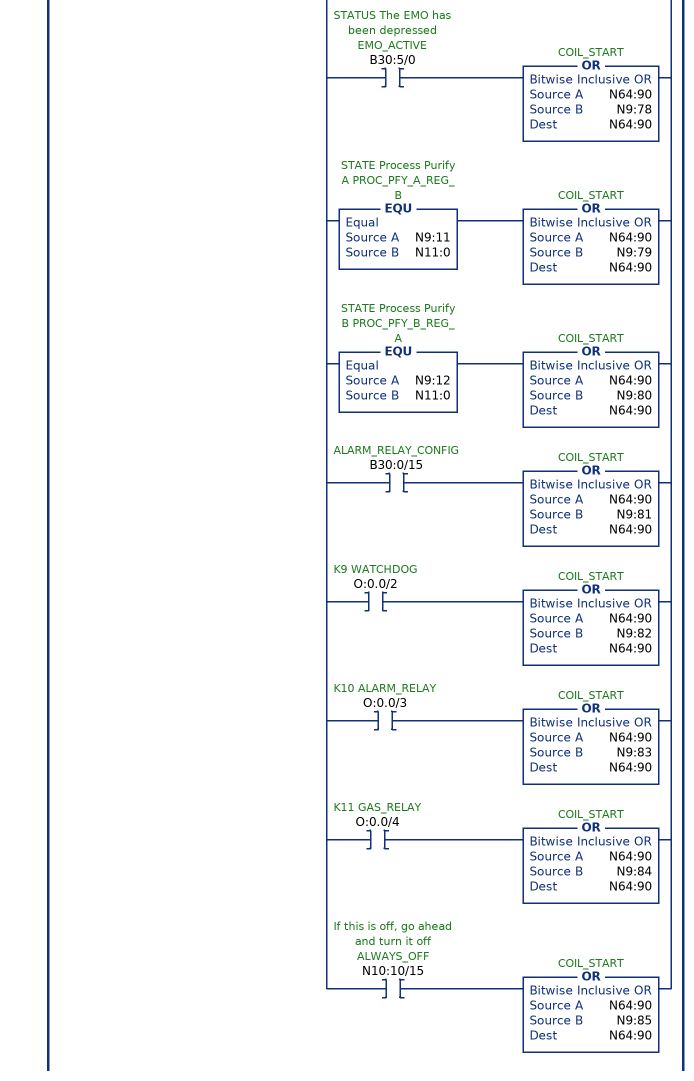
% Rung: 18 %
SOR EQU C5:19.ACC 0 XIO B3:0/3 BST MOV 0 N64:90 NXB XIC T4:153/EN OR N64:90 N9:70 N64:90 NXB XIC N10:16/0 OR N64:90 N9:71 N64:90 NXB XIC B34:2/0 OR N64:90 N9:72 N64:90 NXB XIC N12:4/2 OR N64:90 N9:73 N64:90 NXB BST XIC N10:16/1 NXB XIC B34:2/1 NXB XIC N12:4/3 BND OR N64:90 N9:74 N64:90 NXB EQU N10:0 N9:1 OR N64:90 N9:75 N64:90 NXB EQU N12:0 N9:23 OR N64:90 N9:76 N64:90 NXB XIC B34:0/8 OR N64:90 N9:77 N64:90 NXB XIC B30:5/0 OR N64:90 N9:78 N64:90 NXB EQU N9:11 N11:0 OR N64:90 N9:79 N64:90 NXB EQU N9:12 N11:0 OR N64:90 N9:80 N64:90 NXB XIC B30:0/15 OR N64:90 N9:81 N64:90 NXB XIC O:0.0/2 OR N64:90 N9:82 N64:90 NXB XIC O:0.0/3 OR N64:90 N9:83 N64:90 NXB XIC O:0.0/4 OR N64:90 N9:84 N64:90 NXB XIC N10:10/15 OR N64:90 N9:85 N64:90 BND EOR
%   C5:19  MODBUS_COIL_CTR %
%   B3:0/3  MODBUS_TEST %
%   N64:90  COIL_START %
%   T4:153  MB_HEARTBEAT_ON %
%   N9:70  BIT_0 %
%   N10:16/0  ACTIVE_SYSTEM_ALARM %
%   N9:71  BIT_1 %
%   B34:2/0  ACTIVE_REGEN_ALARM %
%   N9:72  BIT_2 %
%   N12:4/2  ACTIVE_PURIFY_ALARM %
%   N9:73  BIT_3 %
%   N10:16/1  SYSTEM_WARNING_FLAG %
%   B34:2/1  ACTIVE_REGEN_WARNING %
%   N12:4/3  ACTIVE_PURIFY_WARN %
%   N9:74  BIT_4 %
%   N10:0  SYSTEM_STATE  "STATE The current state of the system" %
%   N9:1  SYSTEM_STANDBY  "STATE System Process" %
%   N9:75  BIT_5 %
%   N12:0  PURIFY_STATE  "STATE The current state of the purify process" %
%   N9:23  PURIFY_MANUAL_HOLD  "STATE Purify Manual Hold" %
%   N9:76  BIT_6 %
%   B34:0/8  SET_REGEN_HOLD %
%   N9:77  BIT_7 %
%   B30:5/0  EMO_ACTIVE  "STATUS The EMO has been depressed" %
%   N9:78  BIT_8 %
%   N9:11  PROC_PFY_A_REG_B  "STATE Process Purify A" %
%   N11:0  PROC_STATE  "STATE The current state of the process" %
%   N9:79  BIT_9 %
%   N9:12  PROC_PFY_B_REG_A  "STATE Process Purify B" %
%   N9:80  BIT_10 %
%   B30:0/15  ALARM_RELAY_CONFIG %
%   N9:81  BIT_11 %
%   O:0.0/2  WATCHDOG  "K9" %
%   N9:82  BIT_12 %
%   O:0.0/3  ALARM_RELAY  "K10" %
%   N9:83  BIT_13 %
%   O:0.0/4  GAS_RELAY  "K11" %
%   N9:84  BIT_14 %
%   N10:10/15  ALWAYS_OFF  "If this is off, go ahead and turn it off" %
%   N9:85  BIT_15 %

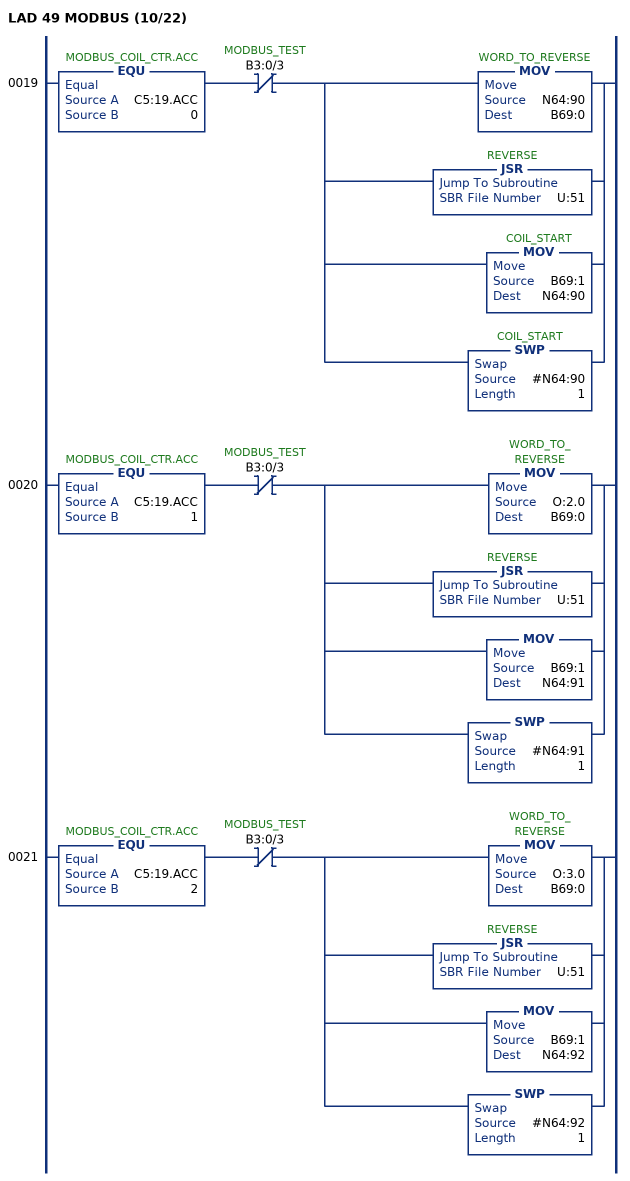
% Rung: 19 %
SOR EQU C5:19.ACC 0 XIO B3:0/3 BST MOV N64:90 B69:0 NXB JSR U:51 NXB MOV B69:1 N64:90 NXB SWP #N64:90 1 BND EOR
%   C5:19  MODBUS_COIL_CTR %
%   B3:0/3  MODBUS_TEST %
%   N64:90  COIL_START %
%   B69:0  WORD_TO_REVERSE %
%   U:51  REVERSE %
%   B69:1  REVERSED_WORD %
% Rung: 20 %
SOR EQU C5:19.ACC 1 XIO B3:0/3 BST MOV O:2.0 B69:0 NXB JSR U:51 NXB MOV B69:1 N64:91 NXB SWP #N64:91 1 BND EOR
%   C5:19  MODBUS_COIL_CTR %
%   B3:0/3  MODBUS_TEST %
%   B69:0  WORD_TO_REVERSE %
%   U:51  REVERSE %
%   B69:1  REVERSED_WORD %
% Rung: 21 %
SOR EQU C5:19.ACC 2 XIO B3:0/3 BST MOV O:3.0 B69:0 NXB JSR U:51 NXB MOV B69:1 N64:92 NXB SWP #N64:92 1 BND EOR
%   C5:19  MODBUS_COIL_CTR %
%   B3:0/3  MODBUS_TEST %
%   B69:0  WORD_TO_REVERSE %
%   U:51  REVERSE %
%   B69:1  REVERSED_WORD %

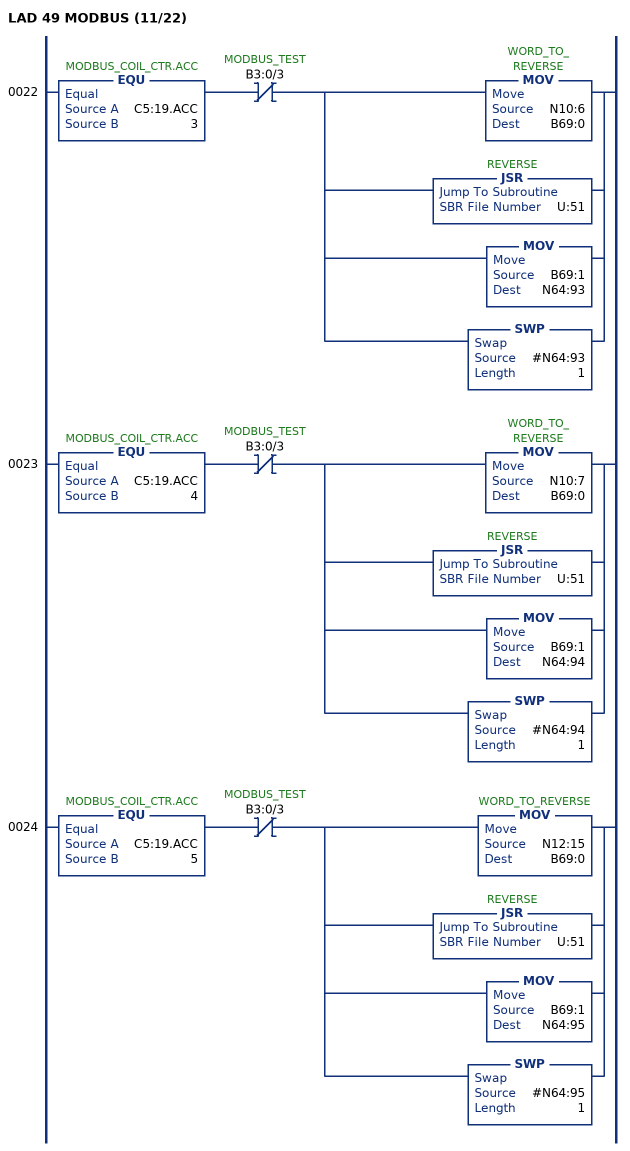
% Rung: 22 %
SOR EQU C5:19.ACC 3 XIO B3:0/3 BST MOV N10:6 B69:0 NXB JSR U:51 NXB MOV B69:1 N64:93 NXB SWP #N64:93 1 BND EOR
%   C5:19  MODBUS_COIL_CTR %
%   B3:0/3  MODBUS_TEST %
%   N10:6  SYSTEM_ALARMS_0  "ALARM System alarms" %
%   B69:0  WORD_TO_REVERSE %
%   U:51  REVERSE %
%   B69:1  REVERSED_WORD %
% Rung: 23 %
SOR EQU C5:19.ACC 4 XIO B3:0/3 BST MOV N10:7 B69:0 NXB JSR U:51 NXB MOV B69:1 N64:94 NXB SWP #N64:94 1 BND EOR
%   C5:19  MODBUS_COIL_CTR %
%   B3:0/3  MODBUS_TEST %
%   N10:7  SYSTEM_ALARMS_1  "ALARM System alarms" %
%   B69:0  WORD_TO_REVERSE %
%   U:51  REVERSE %
%   B69:1  REVERSED_WORD %
% Rung: 24 %
SOR EQU C5:19.ACC 5 XIO B3:0/3 BST MOV N12:15 B69:0 NXB JSR U:51 NXB MOV B69:1 N64:95 NXB SWP #N64:95 1 BND EOR
%   C5:19  MODBUS_COIL_CTR %
%   B3:0/3  MODBUS_TEST %
%   N12:15  PURIFY_ALARMS_0 %
%   B69:0  WORD_TO_REVERSE %
%   U:51  REVERSE %
%   B69:1  REVERSED_WORD %

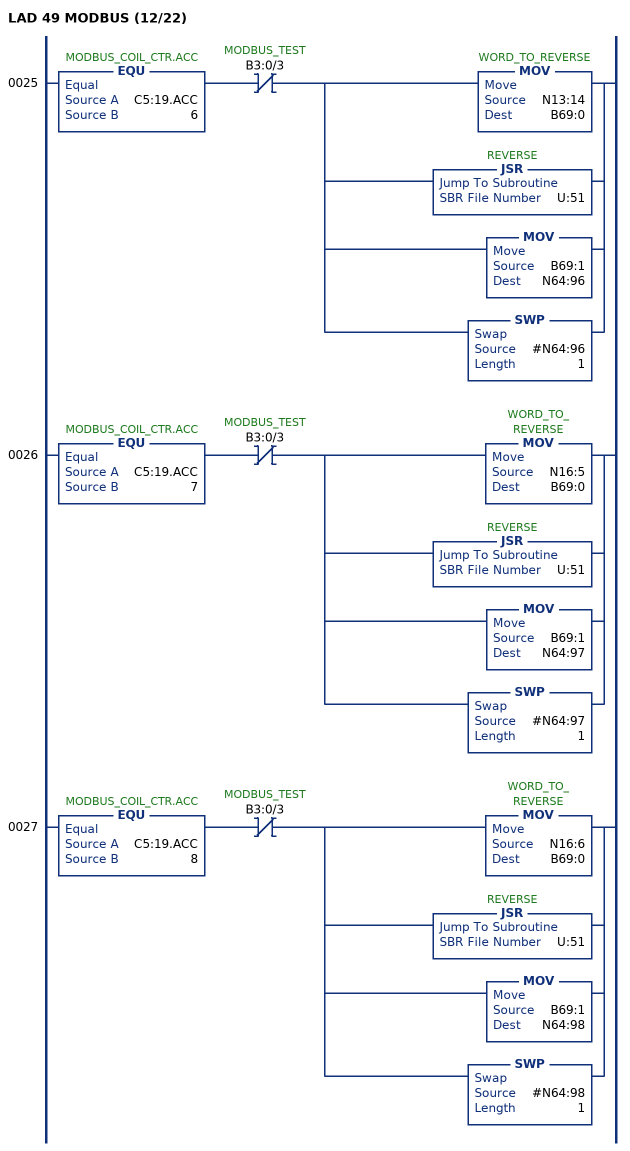
% Rung: 25 %
SOR EQU C5:19.ACC 6 XIO B3:0/3 BST MOV N13:14 B69:0 NXB JSR U:51 NXB MOV B69:1 N64:96 NXB SWP #N64:96 1 BND EOR
%   C5:19  MODBUS_COIL_CTR %
%   B3:0/3  MODBUS_TEST %
%   N13:14  REGEN_ALARMS_0 %
%   B69:0  WORD_TO_REVERSE %
%   U:51  REVERSE %
%   B69:1  REVERSED_WORD %
% Rung: 26 %
SOR EQU C5:19.ACC 7 XIO B3:0/3 BST MOV N16:5 B69:0 NXB JSR U:51 NXB MOV B69:1 N64:97 NXB SWP #N64:97 1 BND EOR
%   C5:19  MODBUS_COIL_CTR %
%   B3:0/3  MODBUS_TEST %
%   N16:5  ADS_A_REGEN_ALARMS_0  "ALARM ADS A Alarms" %
%   B69:0  WORD_TO_REVERSE %
%   U:51  REVERSE %
%   B69:1  REVERSED_WORD %
% Rung: 27 %
SOR EQU C5:19.ACC 8 XIO B3:0/3 BST MOV N16:6 B69:0 NXB JSR U:51 NXB MOV B69:1 N64:98 NXB SWP #N64:98 1 BND EOR
%   C5:19  MODBUS_COIL_CTR %
%   B3:0/3  MODBUS_TEST %
%   N16:6  ADS_A_PURIFY_ALARMS  "ALARM ADS A Alarms" %
%   B69:0  WORD_TO_REVERSE %
%   U:51  REVERSE %
%   B69:1  REVERSED_WORD %

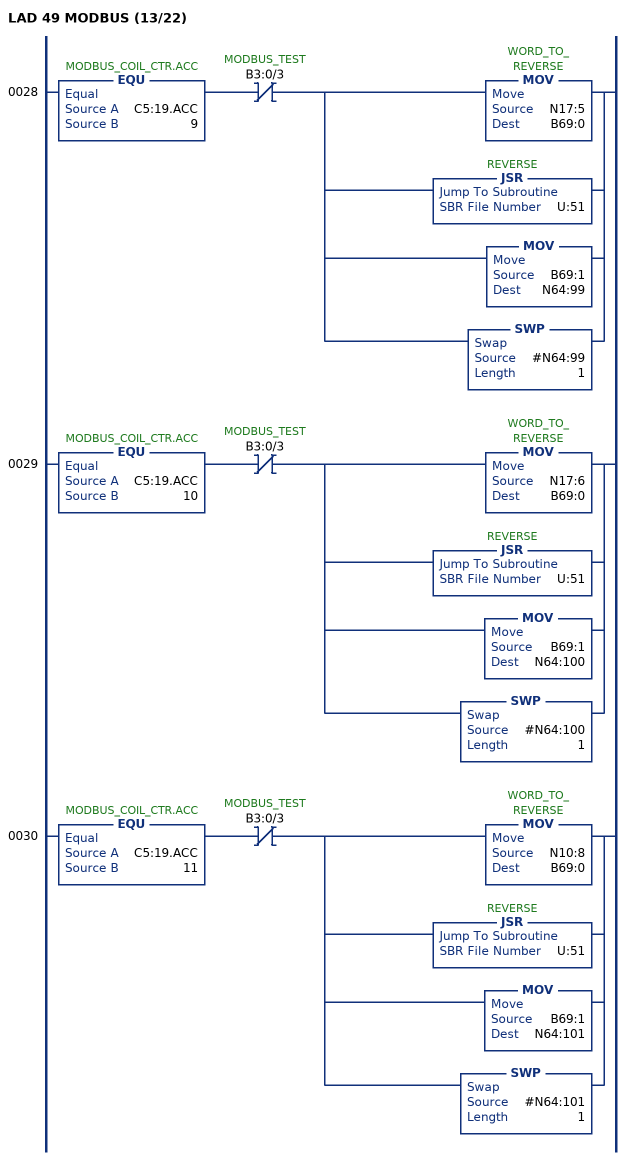
% Rung: 28 %
SOR EQU C5:19.ACC 9 XIO B3:0/3 BST MOV N17:5 B69:0 NXB JSR U:51 NXB MOV B69:1 N64:99 NXB SWP #N64:99 1 BND EOR
%   C5:19  MODBUS_COIL_CTR %
%   B3:0/3  MODBUS_TEST %
%   N17:5  ADS_B_REGEN_ALARMS_0  "ALARM Alarm bits" %
%   B69:0  WORD_TO_REVERSE %
%   U:51  REVERSE %
%   B69:1  REVERSED_WORD %
% Rung: 29 %
SOR EQU C5:19.ACC 10 XIO B3:0/3 BST MOV N17:6 B69:0 NXB JSR U:51 NXB MOV B69:1 N64:100 NXB SWP #N64:100 1 BND EOR
%   C5:19  MODBUS_COIL_CTR %
%   B3:0/3  MODBUS_TEST %
%   N17:6  ADS_B_PURIFY_ALARMS  "ALARM ADS B Alarms" %
%   B69:0  WORD_TO_REVERSE %
%   U:51  REVERSE %
%   B69:1  REVERSED_WORD %
% Rung: 30 %
SOR EQU C5:19.ACC 11 XIO B3:0/3 BST MOV N10:8 B69:0 NXB JSR U:51 NXB MOV B69:1 N64:101 NXB SWP #N64:101 1 BND EOR
%   C5:19  MODBUS_COIL_CTR %
%   B3:0/3  MODBUS_TEST %
%   N10:8  SYSTEM_WARNINGS_0  "WARNING System Warnings" %
%   B69:0  WORD_TO_REVERSE %
%   U:51  REVERSE %
%   B69:1  REVERSED_WORD %

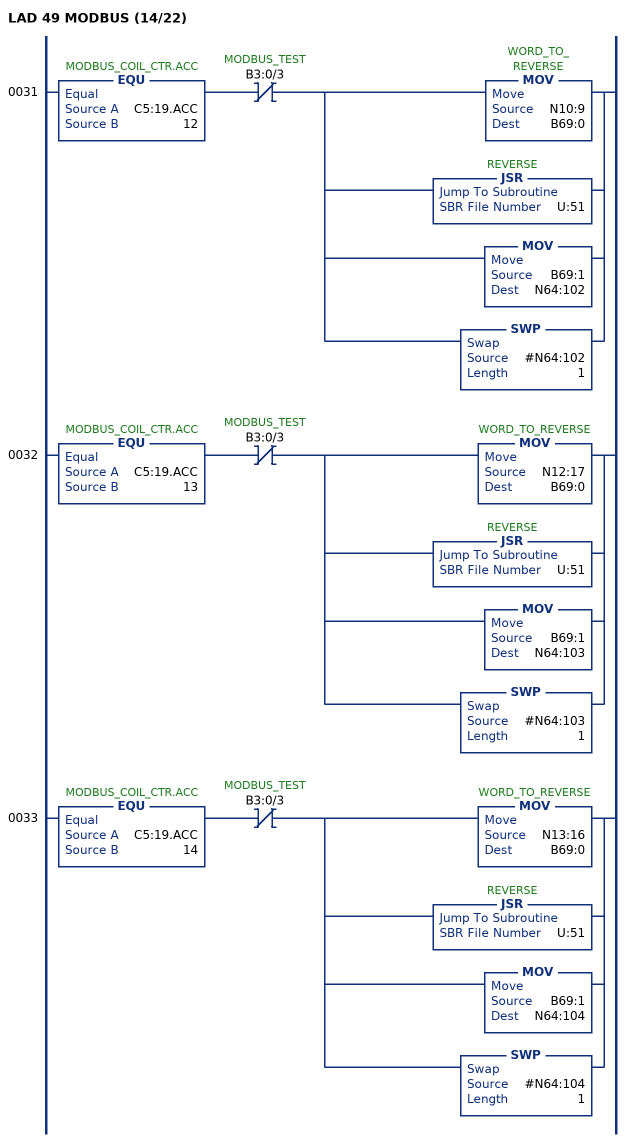
% Rung: 31 %
SOR EQU C5:19.ACC 12 XIO B3:0/3 BST MOV N10:9 B69:0 NXB JSR U:51 NXB MOV B69:1 N64:102 NXB SWP #N64:102 1 BND EOR
%   C5:19  MODBUS_COIL_CTR %
%   B3:0/3  MODBUS_TEST %
%   N10:9  SYSTEM_WARNINGS_1  "WARNING System Warnings" %
%   B69:0  WORD_TO_REVERSE %
%   U:51  REVERSE %
%   B69:1  REVERSED_WORD %
% Rung: 32 %
SOR EQU C5:19.ACC 13 XIO B3:0/3 BST MOV N12:17 B69:0 NXB JSR U:51 NXB MOV B69:1 N64:103 NXB SWP #N64:103 1 BND EOR
%   C5:19  MODBUS_COIL_CTR %
%   B3:0/3  MODBUS_TEST %
%   N12:17  PURIFY_WARNINGS_0 %
%   B69:0  WORD_TO_REVERSE %
%   U:51  REVERSE %
%   B69:1  REVERSED_WORD %
% Rung: 33 %
SOR EQU C5:19.ACC 14 XIO B3:0/3 BST MOV N13:16 B69:0 NXB JSR U:51 NXB MOV B69:1 N64:104 NXB SWP #N64:104 1 BND EOR
%   C5:19  MODBUS_COIL_CTR %
%   B3:0/3  MODBUS_TEST %
%   N13:16  REGEN_WARNINGS_0 %
%   B69:0  WORD_TO_REVERSE %
%   U:51  REVERSE %
%   B69:1  REVERSED_WORD %

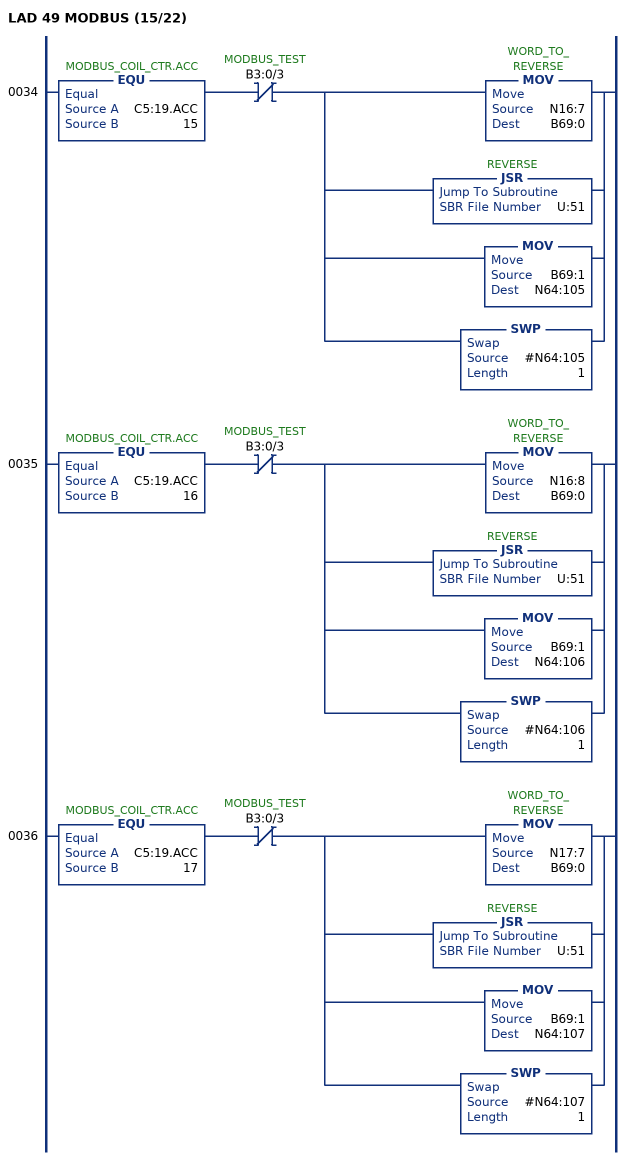
% Rung: 34 %
SOR EQU C5:19.ACC 15 XIO B3:0/3 BST MOV N16:7 B69:0 NXB JSR U:51 NXB MOV B69:1 N64:105 NXB SWP #N64:105 1 BND EOR
%   C5:19  MODBUS_COIL_CTR %
%   B3:0/3  MODBUS_TEST %
%   N16:7  ADS_A_REGEN_WARN_0  "WARNING ADS A Warnings" %
%   B69:0  WORD_TO_REVERSE %
%   U:51  REVERSE %
%   B69:1  REVERSED_WORD %
% Rung: 35 %
SOR EQU C5:19.ACC 16 XIO B3:0/3 BST MOV N16:8 B69:0 NXB JSR U:51 NXB MOV B69:1 N64:106 NXB SWP #N64:106 1 BND EOR
%   C5:19  MODBUS_COIL_CTR %
%   B3:0/3  MODBUS_TEST %
%   N16:8  ADS_A_PURIFY_WARNS  "WARNING ADS A Warnings" %
%   B69:0  WORD_TO_REVERSE %
%   U:51  REVERSE %
%   B69:1  REVERSED_WORD %
% Rung: 36 %
SOR EQU C5:19.ACC 17 XIO B3:0/3 BST MOV N17:7 B69:0 NXB JSR U:51 NXB MOV B69:1 N64:107 NXB SWP #N64:107 1 BND EOR
%   C5:19  MODBUS_COIL_CTR %
%   B3:0/3  MODBUS_TEST %
%   N17:7  ADS_B_REGEN_WARN_0  "WARNING Warning bits" %
%   B69:0  WORD_TO_REVERSE %
%   U:51  REVERSE %
%   B69:1  REVERSED_WORD %

